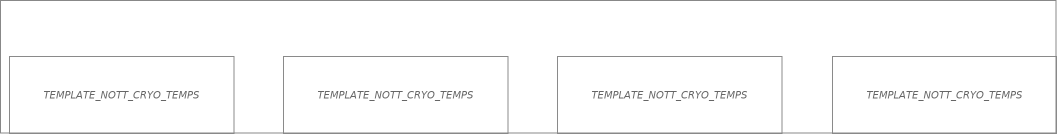
VISUALIZATION GUI_CRYO_TEMPS  // 1057x134
    Frame (9,56 225x78)
        shows TEMPLATE_NOTT_CRYO_TEMPS(m_instance := MAIN.not_cryo_ctrl.temp_1)
    Frame (283,56 225x78)
        shows TEMPLATE_NOTT_CRYO_TEMPS(m_instance := MAIN.not_cryo_ctrl.temp_2)
    Frame (557,56 225x78)
        shows TEMPLATE_NOTT_CRYO_TEMPS(m_instance := MAIN.not_cryo_ctrl.temp_3)
    Frame (832,56 225x78)
        shows TEMPLATE_NOTT_CRYO_TEMPS(m_instance := MAIN.not_cryo_ctrl.temp_4)
END_VISUALIZATION

(* stored: Version 1.1.0.1, ProductVersion 3.1.4024.15
   Visu GUI_CRYO_TEMPS: Id {efd10832-e64f-45a1-8f81-a350470e95a3} *)
